FUNCTION_BLOCK FB_Antriebe
VAR
	Antrieb_Band_1  : FB_Motor;
    Antrieb_Band_2	: FB_Motor;
    Antrieb_Band_3	: FB_Motor;
    Antrieb_Bohrer	: FB_Motor;
    Antrieb_BW_zurueck	: FB_Motor;
    Antrieb_BW_vor	:	FB_Motor;
	FB_Automatik_inst : FB_Autoamtikablauf;
END_VAR

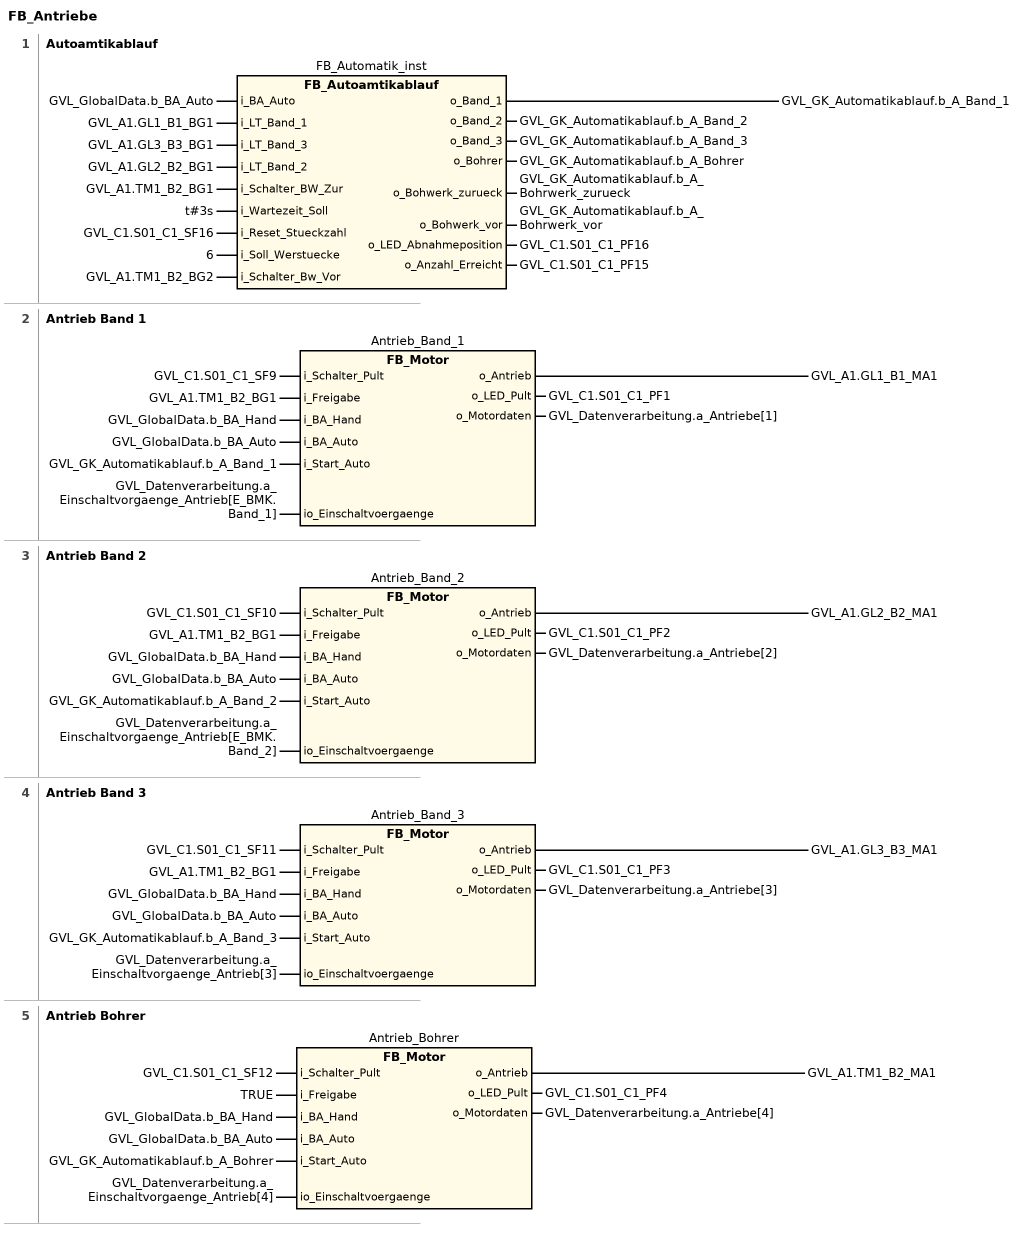
// NETWORK 1: Autoamtikablauf
FB_Automatik_inst(
    i_BA_Auto := GVL_GlobalData.b_BA_Auto,
    i_LT_Band_1 := GVL_A1.GL1_B1_BG1,
    i_LT_Band_3 := GVL_A1.GL3_B3_BG1,
    i_LT_Band_2 := GVL_A1.GL2_B2_BG1,
    i_Schalter_BW_Zur := GVL_A1.TM1_B2_BG1,
    i_Wartezeit_Soll := t#3s,
    i_Reset_Stueckzahl := GVL_C1.S01_C1_SF16,
    i_Soll_Werstuecke := 6,
    i_Schalter_Bw_Vor := GVL_A1.TM1_B2_BG2,
    o_Band_2 => GVL_GK_Automatikablauf.b_A_Band_2,
    o_Band_3 => GVL_GK_Automatikablauf.b_A_Band_3,
    o_Bohrer => GVL_GK_Automatikablauf.b_A_Bohrer,
    o_Bohwerk_zurueck => GVL_GK_Automatikablauf.b_A_Bohrwerk_zurueck,
    o_Bohwerk_vor => GVL_GK_Automatikablauf.b_A_Bohrwerk_vor,
    o_LED_Abnahmeposition => GVL_C1.S01_C1_PF16,
    o_Anzahl_Erreicht => GVL_C1.S01_C1_PF15); // FB_Autoamtikablauf
GVL_GK_Automatikablauf.b_A_Band_1 := FB_Automatik_inst.o_Band_1;

// NETWORK 2: Antrieb Band 1
Antrieb_Band_1(
    i_Schalter_Pult := GVL_C1.S01_C1_SF9,
    i_Freigabe := GVL_A1.TM1_B2_BG1,
    i_BA_Hand := GVL_GlobalData.b_BA_Hand,
    i_BA_Auto := GVL_GlobalData.b_BA_Auto,
    i_Start_Auto := GVL_GK_Automatikablauf.b_A_Band_1,
    io_Einschaltvoergaenge := GVL_Datenverarbeitung.a_Einschaltvorgaenge_Antrieb[E_BMK.Band_1],
    o_LED_Pult => GVL_C1.S01_C1_PF1,
    o_Motordaten => GVL_Datenverarbeitung.a_Antriebe[1]); // FB_Motor
GVL_A1.GL1_B1_MA1 := Antrieb_Band_1.o_Antrieb;

// NETWORK 3: Antrieb Band 2
Antrieb_Band_2(
    i_Schalter_Pult := GVL_C1.S01_C1_SF10,
    i_Freigabe := GVL_A1.TM1_B2_BG1,
    i_BA_Hand := GVL_GlobalData.b_BA_Hand,
    i_BA_Auto := GVL_GlobalData.b_BA_Auto,
    i_Start_Auto := GVL_GK_Automatikablauf.b_A_Band_2,
    io_Einschaltvoergaenge := GVL_Datenverarbeitung.a_Einschaltvorgaenge_Antrieb[E_BMK.Band_2],
    o_LED_Pult => GVL_C1.S01_C1_PF2,
    o_Motordaten => GVL_Datenverarbeitung.a_Antriebe[2]); // FB_Motor
GVL_A1.GL2_B2_MA1 := Antrieb_Band_2.o_Antrieb;

// NETWORK 4: Antrieb Band 3
Antrieb_Band_3(
    i_Schalter_Pult := GVL_C1.S01_C1_SF11,
    i_Freigabe := GVL_A1.TM1_B2_BG1,
    i_BA_Hand := GVL_GlobalData.b_BA_Hand,
    i_BA_Auto := GVL_GlobalData.b_BA_Auto,
    i_Start_Auto := GVL_GK_Automatikablauf.b_A_Band_3,
    io_Einschaltvoergaenge := GVL_Datenverarbeitung.a_Einschaltvorgaenge_Antrieb[3],
    o_LED_Pult => GVL_C1.S01_C1_PF3,
    o_Motordaten => GVL_Datenverarbeitung.a_Antriebe[3]); // FB_Motor
GVL_A1.GL3_B3_MA1 := Antrieb_Band_3.o_Antrieb;

// NETWORK 5: Antrieb Bohrer
Antrieb_Bohrer(
    i_Schalter_Pult := GVL_C1.S01_C1_SF12,
    i_Freigabe := TRUE,
    i_BA_Hand := GVL_GlobalData.b_BA_Hand,
    i_BA_Auto := GVL_GlobalData.b_BA_Auto,
    i_Start_Auto := GVL_GK_Automatikablauf.b_A_Bohrer,
    io_Einschaltvoergaenge := GVL_Datenverarbeitung.a_Einschaltvorgaenge_Antrieb[4],
    o_LED_Pult => GVL_C1.S01_C1_PF4,
    o_Motordaten => GVL_Datenverarbeitung.a_Antriebe[4]); // FB_Motor
GVL_A1.TM1_B2_MA1 := Antrieb_Bohrer.o_Antrieb;

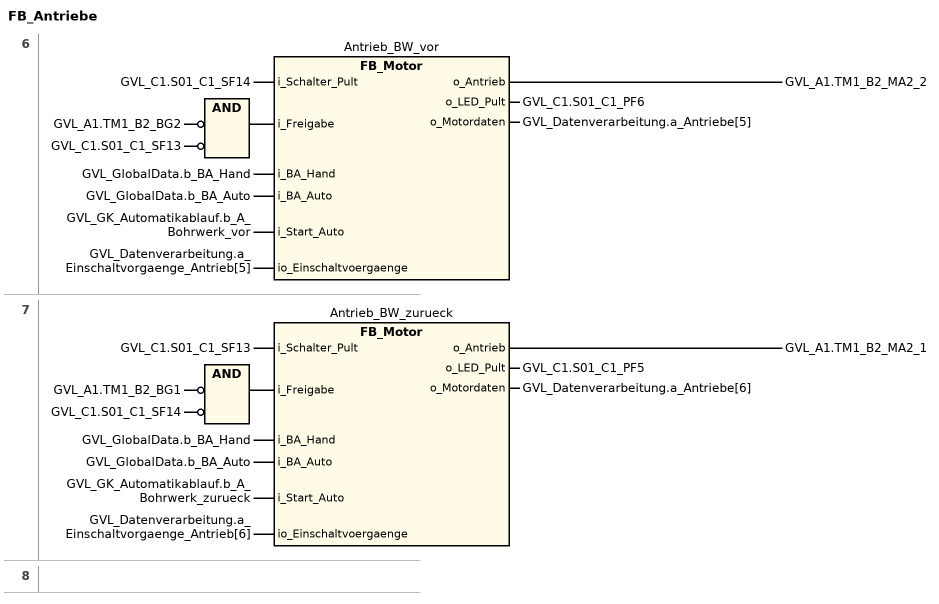
// NETWORK 6
Antrieb_BW_vor(
    i_Schalter_Pult := GVL_C1.S01_C1_SF14,
    i_Freigabe := NOT GVL_A1.TM1_B2_BG2 AND NOT GVL_C1.S01_C1_SF13,
    i_BA_Hand := GVL_GlobalData.b_BA_Hand,
    i_BA_Auto := GVL_GlobalData.b_BA_Auto,
    i_Start_Auto := GVL_GK_Automatikablauf.b_A_Bohrwerk_vor,
    io_Einschaltvoergaenge := GVL_Datenverarbeitung.a_Einschaltvorgaenge_Antrieb[5],
    o_LED_Pult => GVL_C1.S01_C1_PF6,
    o_Motordaten => GVL_Datenverarbeitung.a_Antriebe[5]); // FB_Motor
GVL_A1.TM1_B2_MA2_2 := Antrieb_BW_vor.o_Antrieb;

// NETWORK 7
Antrieb_BW_zurueck(
    i_Schalter_Pult := GVL_C1.S01_C1_SF13,
    i_Freigabe := NOT GVL_A1.TM1_B2_BG1 AND NOT GVL_C1.S01_C1_SF14,
    i_BA_Hand := GVL_GlobalData.b_BA_Hand,
    i_BA_Auto := GVL_GlobalData.b_BA_Auto,
    i_Start_Auto := GVL_GK_Automatikablauf.b_A_Bohrwerk_zurueck,
    io_Einschaltvoergaenge := GVL_Datenverarbeitung.a_Einschaltvorgaenge_Antrieb[6],
    o_LED_Pult => GVL_C1.S01_C1_PF5,
    o_Motordaten => GVL_Datenverarbeitung.a_Antriebe[6]); // FB_Motor
GVL_A1.TM1_B2_MA2_1 := Antrieb_BW_zurueck.o_Antrieb;

// NETWORK 8

END_FUNCTION_BLOCK

(* stored: Version 1.1.0.1, ProductVersion 3.1.4024.12
   POU FB_Antriebe: Id {1a6ad35d-99cd-4d7a-95b3-d72048b9e669}, SpecialFunc None *)
